PROGRAM MAIN
VAR
	iCounter : INT;
	bToggle: BOOL;
	bReset: BOOL;
	stext : STRING := 'Start';
	
	
	fbAlarmingEx	: AlarmingEx;
	
	bAlarm 		: BOOL;
	iAlarm		: INT;
	
	stStruct1		: ST_MyStruct;
END_VAR


IF bToggle THEN
	iCounter := (iCounter+1 ) MOD 1000;
	sText := 'Start';
	IF iCounter = 0 THEN
		bToggle := FALSE;
	END_IF
ELSE
	sText := 'Stop';
	(*
	IF bReset THEN
		bReset := FALSE;
		iCounter := 0;
	END_IF*)

END_IF

Alarming();
fbAlarmingEx();

END_PROGRAM

(* stored: Version 1.1.0.1, ProductVersion 3.1.4024.12
   POU MAIN: Id {2fb61292-a0a1-4762-9537-cc681792ecee}, SpecialFunc None *)
